       #FB_STATE_TCP_RECONNECTING:
         REGION FB_STATE_TCP_RECONNECTING
           IF #tempTsendcStatus = #TSENDC_EST_OK THEN
             #statErrorAutoCleared := FALSE;
             // Update edge detection
             #statPublishOld := #tempPublish;
             #statSubscribeOld := #tempSubscribe;
             #statUnsubscribeOld := #tempUnsubscribe;
             //Monitor Connection
             #statFBState := #FB_STATE_OPERATING_MONITOR_TCP;
             // Begin MQTT Connection
             #statMqttConnectState := #MQTT_CONNECT_STATE_BUILD_PAKET;
           END_IF;
         END_REGION FB_STATE_TCP_RECONNECTING
       #FB_STATE_DISABLING: // Disabling active
         REGION DISABLING FB
           //  Disabling, e.g. closing connections, etc.
           // When disabling is complete the bit #statDisablingCompleted must be set
           // When MQTT is connected, send disconnect
           IF #statMqttConnectState = #MQTT_CONNECT_STATE_CONNECTED THEN
             IF #statTsendcReq = TRUE THEN
               //Interrupt any existing send jobs
               #statTsendcReq := FALSE;
             ELSE
               // INIT
               #statSendBufferPos := 0;
               //Build fixed Header
               //Message Type
               #statSendBuffer[#statSendBufferPos] := #MQTT_MSG_TYPE_DISCONNECT;
               #statSendBufferPos += 1;
               //Remaining Length (must be O)
               #statSendBuffer[#statSendBufferPos] := #REMAINIG_LEN_0;
               #statSendBufferPos += 1;
               //send request
               #statTsendcLen := #statSendBufferPos;
               #statTsendcReq := TRUE;
               #statMqttConnectState := #MQTT_CONNECT_STATE_DISCONNECTED;
             END_IF;
           ELSE
             //Disable TCP Connection
             #statTsendcReq := FALSE;
             #statTsendcEnable := FALSE;
             #statEnableTimerCommandWatchdog := TRUE;
           END_IF;
           // When TCP connection is closed
           IF #tempTsendcStatus = #TSENDC_DISCONNECTED THEN
             #statEnableTimerCommandWatchdog := FALSE;
             #statDisablingCompleted := TRUE;
           ELSIF #instTimerCommandWatchdog.Q THEN
             #statEnableTimerCommandWatchdog := FALSE;
             #statDisablingCompleted := TRUE;
           END_IF;
         END_REGION DISABLING FB
       ELSE // Undefined state in state machine reached
         #statStatus := #ERR_UNDEFINED_STATE;
         #statErrorUserCleared := TRUE;
     END_CASE;
   END_REGION STATE_MACHINE

   REGION OUTPUTS
     // Write outputs
     IF (#statDisablingCompleted = TRUE) THEN
       // Reset outputs if disabling completed
       #statValid := FALSE;
       #statBusy := FALSE;
       #statError := FALSE;
       #statDone := FALSE;
       #statErrorUserCleared := FALSE;
       #statErrorAutoCleared := FALSE;
       #statStatus := #STATUS_NO_CALL;
       // Reset application specific outputs
       #statRcvMsgStatus := #MSG_DECODE_STATUS_NO_NEW_MSG;
       #statRcvMsgDataLen := 0;

     ELSIF (#statErrorUserCleared = TRUE) AND (#statError = FALSE) THEN
       // Error can only be cleared by user; rising edge at enable input is needed to continue 
       #statValid := FALSE;
       #statBusy := FALSE;
       #statDone := FALSE;
       #statError := TRUE;
       // Write diagnostics
       #diagnostics.status := #statStatus;
       #diagnostics.subfunctionStatus := #statSubfunctionStatus;
       #diagnostics.stateNumber := #statFBErrorState;
       // execution aborted --> set state no processing
       #statTsendcEnable := FALSE; // Terminate Connection, no reason keep it up.
       #statFBState := #FB_STATE_NO_PROCESSING;
       #statMqttConnectState := #MQTT_CONNECT_STATE_NO_PROCESSING;
       #statMqttCommandState := #MQTT_COMMAND_STATE_NO_PROCESSING;
       #statRcvMsgDecodeState := #MSG_DECODE_STATE_NO_PROCESSING;

     ELSIF (#statErrorAutoCleared = TRUE) AND (#statError = FALSE) THEN
       // Error can be reset by FB automatically
       #statValid := FALSE;
       #statBusy := TRUE;
       #statError := TRUE;
       #statDone := FALSE;

       // Write diagnostics
       #diagnostics.status := #statStatus;
       #diagnostics.subfunctionStatus := #statSubfunctionStatus;
       #diagnostics.stateNumber := #statFBErrorState;
       // Handling of autocleared error
       CASE #statStatus OF
           //Just signal error and reset autocleared error afterwards.
         #ERR_MQTT_PAKET_ID_INVALID, #ERR_MQTT_SUBACK_FAILURE, #ERR_MQTT_CONNECT_TIMEOUT,
         #ERR_MQTT_COMMAND_SEND_TIMEOUT, #ERR_MQTT_COMMAND_MULTIPLE_INPUT, #ERR_CNT_EXCEEDS_ARRAY_DIMENSION,
         #ERR_MQTT_COMMAND_PUBLISH_TOPIC_INVALID, #ERR_QOS_INVALID, #ERR_MQTT_COMMAND_SUBSCRIBE_TOPIC_INVALID:
           #statErrorAutoCleared := FALSE;

         ELSE  // Statement section ELSE
           ;
       END_CASE;

     ELSIF (#statErrorAutoCleared = FALSE) AND (#statErrorUserCleared = FALSE) AND (#statError = TRUE) THEN
       // If autocleared error is acknowledged
       #statValid := TRUE;
       #statBusy := TRUE;
       #statError := FALSE;
       #statDone := FALSE;

       //   this line  more detailed status information is used instead of "#STATUS_SUBSEQUENT_CALL"
       CASE #statStatus OF
         #ERR_TCP_RECONNECTING, #ERR_MQTT_CONNECT_TIMEOUT:  // Reconnecting ok, start Mqtt reconnnect
           //set status
           #statStatus := #STATUS_MQTT_CONNECTING;
           //in the following status codes status stays connected. 
         #ERR_MQTT_PAKET_ID_INVALID, #ERR_MQTT_SUBACK_FAILURE, #ERR_MQTT_COMMAND_SEND_TIMEOUT,
         #ERR_MQTT_COMMAND_MULTIPLE_INPUT, #ERR_CNT_EXCEEDS_ARRAY_DIMENSION, #ERR_MQTT_COMMAND_PUBLISH_TOPIC_INVALID,
         #ERR_QOS_INVALID, #ERR_MQTT_COMMAND_SUBSCRIBE_TOPIC_INVALID:
           #statStatus := #STATUS_MQTT_CONNECTED;
         ELSE  // Statement section ELSE
           ;
       END_CASE;
     END_IF;

     // Write static values to outputs
     #valid := #statValid;
     #busy := #statBusy;
     #error := #statError;
     #status := #statStatus;
     //block sets ENO automatically:
     //ENO := TRUE;
     //Write application specific static values to outputs
     #done := #statDone;
     #receivedMsgStatus := #statRcvMsgStatus;
     #receivedMsgDataLen := #statRcvMsgDataLen;
   END_REGION OUTPUTS
END_FUNCTION_BLOCK

// folder: LMQTT/Utilities

FUNCTION "LMQTT_ConvertToUtf8" : Void   // FC6, SCL
TITLE = LMQTT_ConvertToUtf8
{ S7_Optimized_Access := 'TRUE' }
AUTHOR : SIEMENS
FAMILY : LMQTT
VERSION : 1.0
// Function to convert a WCHAR to a UTF-8 conformant byte sequence
   VAR_INPUT
      character : WChar;   // Character that shall be converted to UTF-8
   END_VAR
   VAR_OUTPUT
      convertedUtf8 : DWord;   // UTF-8 conformant byte sequence. B0 stores first Byte, B1 second and B2 third Byte. B3 is not used
      bytesUsed : USInt;   // Amount of Bytes converted. Ranges from 1 to 3.
      error : Bool;   // TRUE: An error occurred during the execution of the FC
      status : Word;   // 16#0000 - 16#7FFF: Status of the FC, 16#8000 - 16#FFFF: Error identification
   END_VAR
   VAR_TEMP
      tempStatus : Word;   // temp value for output 'status'
      tempConvertedUtf8 : DWord;   // temp value for output 'convertedUtf8'
      tempBytesUsed : USInt;   // temp value for output 'bytesUsed'
      tempCharacter : WChar;   // temp value for input 'character'
   END_VAR
   // Ret_Val : No return for this FC - see error and status output
   VAR CONSTANT
      STATUS_NO_ERROR : Word := 16#0000;   // no error status
      STATUS_EXECUTION_FINISHED : Word := 16#0000;   // Execution finished without errors
      ERR_UNDEFINED : Word := 16#8000;   // Error due to an undefined case
      USINT_NULL : USInt := 0;   // Init value with 0
      DWORD_NULL : DWord := 16#0000_0000;   // Init value with 0
      EMPTY_WCHAR : WChar := WCHAR#' ';   // Empty WChar for comparison
      BELOW_7F : Word := 16#007F;   // Upper limit for character if only one Byte used
      BELOW_7FF : Word := 16#07FF;   // Upper limit for character if two Byte used
      BELOW_MAX_FFFF : Word := 16#FFFF;   // Upper limit for character if three Byte used
      BYTE_3F : Byte := 16#3F;   // Conversion Value
      BYTE_80 : Byte := 16#80;   // Conversion Value
      BYTE_C0 : Byte := 16#C0;   // Conversion Value
      BYTE_E0 : Byte := 16#E0;   // Conversion Value
      USINT_ONE : USInt := 1;   // Const Value to assign amount of bytes used
      USINT_TWO : USInt := 2;   // Const Value to assign amount of bytes used
      USINT_THREE : USInt := 3;   // Const Value to assign amount of bytes used
   END_VAR
BEGIN
   REGION BLOCK INFO HEADER
       //=============================================================================
       // SIEMENS AG
       // (c)Copyright 2020
       //-----------------------------------------------------------------------------
       // Library:       LMQTT
       // Tested with:   CPU 1516-3 PN/DP V2.8
       // Engineering:   TIA Portal V16
       // Restrictions:  --
       // Requirements:  --
       // Functionality: Converts a single WChar Character to a valid UTF-8 encoded byte sequence and saves this to a DWord.
       //                The amount of bytes saved is stored in bytesUsed Output.
       //-----------------------------------------------------------------------------
       // Change log table:
       // Version    Date         Expert in charge         Changes applied
       // 03.00.00   01.10.2020   Siemens Online Support   First released version
       //=============================================================================
   END_REGION

   REGION INITIALISATION  
       // Initialize functionality: reset of variables, diagnostics, etc.
       #tempConvertedUtf8 := #DWORD_NULL;
       #tempBytesUsed := #USINT_NULL;
       #tempStatus := #STATUS_NO_ERROR;
       //assign temp value from input:
        #tempCharacter := #character;

   END_REGION

   REGION PROGRAM LOGIC
       // Use this region for application specific code
       IF #tempCharacter = #EMPTY_WCHAR THEN
           //will be only 1 byte occupied
           #tempConvertedUtf8 := WCHAR_TO_DWORD(#tempCharacter);
           #tempBytesUsed := #USINT_ONE;
       ELSIF (WCHAR_TO_WORD(#tempCharacter) <= (#BELOW_7F)) THEN
           //will be only 1 byte occupied
           #tempConvertedUtf8 := WCHAR_TO_DWORD(#tempCharacter);
           #tempBytesUsed := #USINT_ONE;
       ELSIF (WCHAR_TO_WORD(#tempCharacter) <= (#BELOW_7FF)) THEN
           //will be 2 byte occupied
           #tempConvertedUtf8.%B1 := (WCHAR_TO_BYTE(#tempCharacter) AND #BYTE_3F) OR #BYTE_80;
           #tempConvertedUtf8.%B0 := WORD_TO_BYTE(SHR(IN := WCHAR_TO_WORD(#tempCharacter), N := 6)) OR #BYTE_C0;
           #tempBytesUsed := #USINT_TWO;
       ELSIF (WCHAR_TO_WORD(#tempCharacter) <= (#BELOW_MAX_FFFF)) THEN
           //will be 3 byte occupied
           #tempConvertedUtf8.%B2 := (WCHAR_TO_BYTE(#tempCharacter) AND #BYTE_3F) OR #BYTE_80;
           #tempConvertedUtf8.%B1 := (WORD_TO_BYTE(SHR(IN := WCHAR_TO_WORD(#tempCharacter), N := 6)) AND #BYTE_3F) OR #BYTE_80;
           #tempConvertedUtf8.%B0 := WORD_TO_BYTE(SHR(IN := WCHAR_TO_WORD(#tempCharacter), N := 12)) OR #BYTE_E0;
           #tempBytesUsed := #USINT_THREE;
       END_IF;
   END_REGION

   REGION OUTPUTS
       // Write application specific temp values to outputs
       #bytesUsed := #tempBytesUsed;
       #convertedUtf8 := #tempConvertedUtf8;
       // Write error and status
       #error := #tempStatus.%X15;
       #status := #tempStatus;
       // ENO mechanism is not used --> ENO := TRUE;
       ENO := TRUE;
   END_REGION
END_FUNCTION